FUNCTION F_MKS_909 : INT
VAR_INPUT
	stGauge	:	ST_MKS_909;
END_VAR
VAR
END_VAR

(* Converts real pressure to digital voltage for 937A/B *)
IF stGauge.rPress <> 0 THEN
	F_MKS_909 := REAL_TO_INT( (32767/10) * (LOG( stGauge.rPress ) + 10) );
ELSE
	F_MKS_909 := 0;
END_IF

END_FUNCTION

(* stored: Version 1.1.0.1, ProductVersion 3.1.4020.12
   POU F_MKS_909: Id {0f108d56-1826-44ef-b8a5-046ec9eba208}, SpecialFunc None *)
